// TwinCAT 3 PLC project Untitled1
// ProgramVersion: 3.1.4023.0
// libraries:
//   Tc2_Standard, * (Beckhoff Automation GmbH)
//   Tc2_System, * (Beckhoff Automation GmbH)
//   Tc2_Utilities, * (Beckhoff Automation GmbH)
//   Tc3_Module, * (Beckhoff Automation GmbH)
// project tree:
//   DUTs/ E_EventType.TcDUT (not stored), ST_Event.TcDUT (not stored)
//   Functions/ Sign.TcPOU (not stored)
//   GVLs/ SimulationVariables.TcGVL (not stored)
//   Main Program/ MAIN.TcPOU
//   / PlcTask.TcTTO (not stored)
//   POUs/ DiscreteIntegrator.TcPOU (not stored), ElectricMotor.TcPOU, EventLogger.TcPOU (not stored), HydraulicCylinder.TcPOU (not stored), OrificeEquation.TcPOU (not stored), PressureBuildUp.TcPOU (not stored), PressureGradient.TcPOU (not stored), Pump.TcPOU (not stored), UpdateEventTimestamptWithSystemTime.TcPOU (not stored)

// ---- Main Program/MAIN.TcPOU
PROGRAM MAIN
VAR
	//stThisIsOurFirstInstanceOfAStructure : ST_Event;
	bBoolean : BOOL := FALSE;
	eEventType1 : E_EventType := E_EventType.Alarm;
	eEventSeverity1 : TcEventSeverity := TcEventSeverity.Error;
	nEventIdentity1 : UDINT := 42;
	sEventText1 : STRING(255) := 'This is halloween';
	EventLogger : EventLogger;
	
///////////////////////////////////////////////////////////////////////////////////////

	//Integrator
	ssMethodType : SINT := 1; 
	Timer : LREAL;
	
	//PressureA
	fbPressure : DiscreteIntegrator;
	fbPressureGradient : PressureGradient;
	Pressure : LREAL;
	
	//Pump
	fbPump : Pump;
	PumpTorque : LREAL;
	PumpFlowRate : LREAL;

	//OrificeEquation
	fbOrificeEquation1 : OrificeEquation;
	fbOrificeEquation2 : OrificeEquation;	
	OrificeFlow: LREAL;

END_VAR

(* IF NOT bBoolean THEN
	UpdateEventTimestamptWithSystemTime(stEvent := stThisIsOurFirstInstanceOfAStructure);
	bBoolean := TRUE;
END_IF *)

IF bBoolean THEN
	EventLogger.AddEvent(eEventType1, eEventSeverity1, nEventIdentity1, sEventText1);
	bBoolean := FALSE;
END_IF

//Timer
Timer := Timer + 0.01;

//PressureGradient
fbPressureGradient(
	TotalVolume := 2.9444E-04,
	BulkModulus := 10000.0,
	FlowrateIn := 60.0,
	FlowrateOut := 20.0
	);

//PressureA
fbPressure(
	ssMethodType := ssMethodType,
	In1 := fbPressureGradient.PressureGradientPascal,
	Out1 => Pressure
	);

//Pump
fbPump(
	MotorSpeedRPM := 413.2,
	PumpDisplacement := 10.6E-6,
	DeltaMaxPressure := 250.0,
	PumpTorque => PumpTorque,
	PumpFlowRate => PumpFlowRate
	);
	
//OrificeEquation1
fbOrificeEquation1(
	PressureOut := 4; 			//Found value from old simulink project, this one goes to the tank i guess
	PressureIn := Pressure;		//Just taken the pressure from the pressureA value		
	Kv := ;
	ValveOpening := ;	
	OrificeFlow => OrificeFlow
	);

END_PROGRAM

// ---- POUs/ElectricMotor.TcPOU
FUNCTION_BLOCK ElectricMotor
VAR_INPUT
	ssMethodType: SINT;
	CylinderSetPosition: LREAL;
	CylinderCurrentPosition: LREAL;
	CylinderCurrentVelocity: LREAL;
END_VAR
VAR_OUTPUT
	MotorSpeedRPM: LREAL;
END_VAR
VAR
	rtb_Sum2: LREAL;
	rtb_IntegralGain: LREAL;
	Integrator_DSTATE: LREAL;
	Integrator_DSTATE_i: LREAL;
END_VAR



CASE ssMethodType OF
    0: 
        (* SystemInitialize for Atomic SubSystem: '<Root>/ElectricMotor' *)
        (* InitializeConditions for DiscreteIntegrator: '<S35>/Integrator' *)
        Integrator_DSTATE := 0.0;
        (* InitializeConditions for DiscreteIntegrator: '<S83>/Integrator' *)
        Integrator_DSTATE_i := 0.0;
        (* End of SystemInitialize for SubSystem: '<Root>/ElectricMotor' *)
    1: 
        (* Outputs for Atomic SubSystem: '<Root>/ElectricMotor' *)
        (* Sum: '<S1>/Sum1' *)
        rtb_Sum2 := CylinderSetPosition - CylinderCurrentPosition;
        (* Gain: '<S32>/Integral Gain' *)
        rtb_IntegralGain := 0.001 * rtb_Sum2;
        (* Sum: '<S44>/Sum' incorporates:
         *  DiscreteIntegrator: '<S35>/Integrator'
         *  Gain: '<S40>/Proportional Gain' *)
        rtb_Sum2 := (5.0 * rtb_Sum2) + Integrator_DSTATE;
        (* Saturate: '<S42>/Saturation' *)

        IF rtb_Sum2 > 0.23 THEN 
            rtb_Sum2 := 0.23;
        ELSIF rtb_Sum2 < -0.23 THEN 
            rtb_Sum2 := -0.23;
        END_IF;

        (* End of Saturate: '<S42>/Saturation' *)
        

        (* Sum: '<S1>/Sum2' *)
        rtb_Sum2 := rtb_Sum2 - CylinderCurrentVelocity;
        (* Outport: '<Root>/MotorSpeedRPM' incorporates:
         *  DiscreteIntegrator: '<S83>/Integrator'
         *  Gain: '<S88>/Proportional Gain'
         *  Sum: '<S92>/Sum' *)
        MotorSpeedRPM := (2000.0 * rtb_Sum2) + Integrator_DSTATE_i;
        (* Update for DiscreteIntegrator: '<S35>/Integrator' *)
        Integrator_DSTATE := (0.001 * rtb_IntegralGain) + Integrator_DSTATE;
        (* Update for DiscreteIntegrator: '<S83>/Integrator' incorporates:
         *  Gain: '<S80>/Integral Gain' *)
        Integrator_DSTATE_i := ((0.01 * rtb_Sum2) * 0.001) + Integrator_DSTATE_i;
        (* End of Outputs for SubSystem: '<Root>/ElectricMotor' *)
END_CASE;

END_FUNCTION_BLOCK
